(* Logix 5000 project; controller axis1 vendor 1 type 14 code 155 rev 20.12; software revision 20.01 *)

TASK MainTask (continuous, watchdog 500 ms) : MainProgram

MODULES
   Local : vendor 1 type 14 code 155 (PointIO 0, rev 20.12)
      Kinetix_350 : vendor 1 type 37 code 27 (Ethernet 192.168.1.7, rev 1.1, MotionDiagnostics RPI 1 ms, MotionSync RPI 2 ms)
       : 1734-IE2V (PointIO 2, rev 3.1, Input RPI 80 ms)
      Discrete_IO : Embedded (PointIO 1, rev 20.11, Output RPI 20 ms)
       : 1734-OE2V (PointIO 3, rev 3.1, Output RPI 80 ms)
       : vendor 1 type 109 code 13 (PointIO 4, rev 3.1, Output RPI 80 ms)
END_MODULES

VAR_GLOBAL   (* controller tags *)
   Axis_1 : AXIS_CIP_DRIVE;
   Kinetix_350_Quick_Start : MOTION_GROUP;
END_VAR

PROGRAM MainProgram   (* main routine MainRoutine *)
VAR
   Axis1_Motion : MOTION_INSTRUCTION;
   MOVE_step0 : MOTION_INSTRUCTION;
   MOVE_step1 : MOTION_INSTRUCTION;
   move_step2 : MOTION_INSTRUCTION;
   MOVE_step3 : MOTION_INSTRUCTION;
   MOVE_step4 : MOTION_INSTRUCTION;
   MOVE_step5 : MOTION_INSTRUCTION;
   MOVE_step6 : MOTION_INSTRUCTION;
   MOVE_step7 : MOTION_INSTRUCTION;
   MOVE_step8 : MOTION_INSTRUCTION;
   MOVE_step9 : MOTION_INSTRUCTION;
   one_shot1 : BOOL;
END_VAR

ROUTINE MainRoutine   (* ladder *)
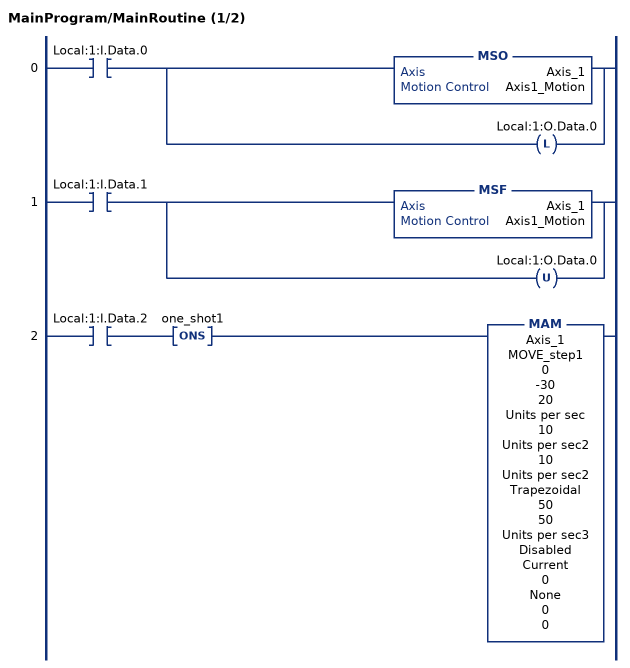
   0: XIC(Local:1:I.Data.0)[MSO(Axis_1,Axis1_Motion) ,OTL(Local:1:O.Data.0) ];
   1: XIC(Local:1:I.Data.1)[MSF(Axis_1,Axis1_Motion) ,OTU(Local:1:O.Data.0) ];
   2: XIC(Local:1:I.Data.2)ONS(one_shot1)MAM(Axis_1,MOVE_step1,0,-30,20,Units per sec,10,Units per sec2,10,Units per sec2,Trapezoidal,50,50,Units per sec3,Disabled,Current,0,None,0,0);
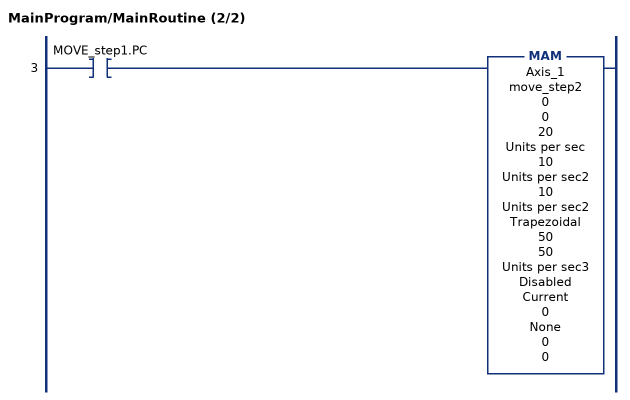
   3: XIC(MOVE_step1.PC)MAM(Axis_1,move_step2,0,0,20,Units per sec,10,Units per sec2,10,Units per sec2,Trapezoidal,50,50,Units per sec3,Disabled,Current,0,None,0,0);
END_ROUTINE
END_PROGRAM
